FUNCTION_BLOCK PLOT_2_CURVES
  {SET_ATTRIBUTE(OpcUa, SERVICE)}
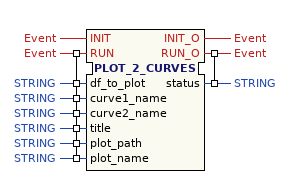
  EVENT_INPUT
    INIT;
    RUN WITH df_to_plot, curve1_name, curve2_name, title, plot_path, plot_name; {SET_ATTRIBUTE(OpcUa, Method)}
  END_EVENT
  EVENT_OUTPUT
    INIT_O;
    RUN_O WITH status;
  END_EVENT
  VAR_INPUT
    df_to_plot : STRING; {SET_ATTRIBUTE(OpcUa, Variable.RUN)}
    curve1_name : STRING; {SET_ATTRIBUTE(OpcUa, Variable.RUN)}
    curve2_name : STRING; {SET_ATTRIBUTE(OpcUa, Variable.RUN)}
    title : STRING; {SET_ATTRIBUTE(OpcUa, Variable.RUN)}
    plot_path : STRING; {SET_ATTRIBUTE(OpcUa, Variable.RUN)}
    plot_name : STRING; {SET_ATTRIBUTE(OpcUa, Variable.RUN)}
  END_VAR
  VAR_OUTPUT
    status : STRING; {SET_ATTRIBUTE(OpcUa, Variable.RUN)}
  END_VAR
END_FUNCTION_BLOCK
